# B&R Automation Studio project Lab2_Conveyor (part 2)

### Stations.var - not listed in the package file held
```iecst
VAR
	Conveyor : Conveyor_typ := (Input:=(Par:=(Accel:=100.0,Speed:=100.0,Decel:=100.0)));
	Ejector : Ejector_typ; (*Interface for the Ejector Station*)
	SwivelArm : SwivelArm_typ;
END_VAR
```

### Program Logical/Distributing/Machine/Ejector (IEC)

#### Cyclic.ld - Cyclic code
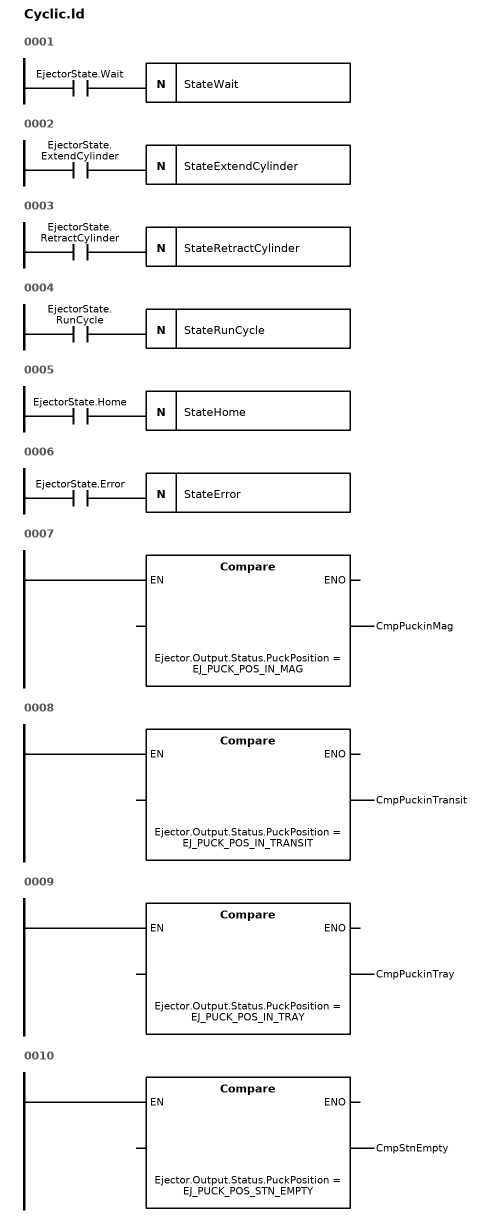
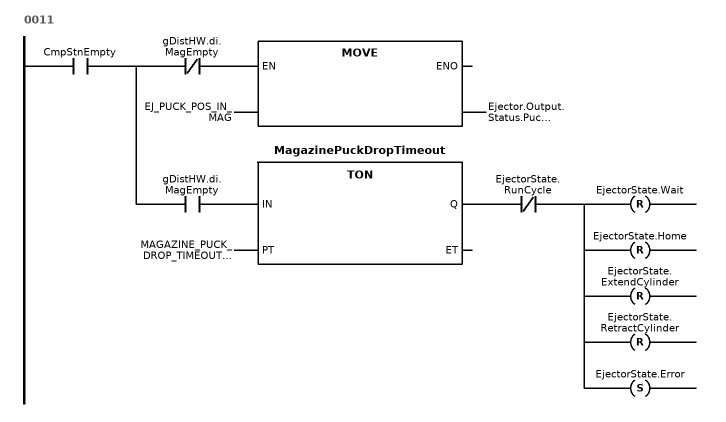
Ladder, written as Structured Text:
```iecst
(*********************************************************************************
 * Copyright: 	B&R Industrial Automation
 * Author:    	Matthew Boyes
 * Created:   	March 8, 2019/12:38 PM
 * Description: 	Task for controlling the operation of the Ejector Station.
 *********************************************************************************)
PROGRAM _CYCLIC
VAR
    _p1 : BOOL;
END_VAR
(* Network 1 *)
IF EjectorState.Wait THEN StateWait; END_IF;

(* Network 2 *)
IF EjectorState.ExtendCylinder THEN StateExtendCylinder; END_IF;

(* Network 3 *)
IF EjectorState.RetractCylinder THEN StateRetractCylinder; END_IF;

(* Network 4 *)
IF EjectorState.RunCycle THEN StateRunCycle; END_IF;

(* Network 5 *)
IF EjectorState.Home THEN StateHome; END_IF;

(* Network 6 *)
IF EjectorState.Error THEN StateError; END_IF;

(* Network 7 *)
CmpPuckinMag := Ejector.Output.Status.PuckPosition = EJ_PUCK_POS_IN_MAG;

(* Network 8 *)
CmpPuckinTransit := Ejector.Output.Status.PuckPosition = EJ_PUCK_POS_IN_TRANSIT;

(* Network 9 *)
CmpPuckinTray := Ejector.Output.Status.PuckPosition = EJ_PUCK_POS_IN_TRAY;

(* Network 10 *)
CmpStnEmpty := Ejector.Output.Status.PuckPosition = EJ_PUCK_POS_STN_EMPTY;

(* Network 11 *)
IF CmpStnEmpty AND NOT gDistHW.di.MagEmpty THEN
    Ejector.Output.Status.PuckPosition := EJ_PUCK_POS_IN_MAG;
END_IF;
MagazinePuckDropTimeout(IN := CmpStnEmpty AND gDistHW.di.MagEmpty, PT := MAGAZINE_PUCK_DROP_TIMEOUT_VALUE);
_p1 := MagazinePuckDropTimeout.Q AND NOT EjectorState.RunCycle;
IF _p1 THEN
    EjectorState.Wait := FALSE;
    EjectorState.Home := FALSE;
    EjectorState.ExtendCylinder := FALSE;
    EjectorState.RetractCylinder := FALSE;
    EjectorState.Error := TRUE;
END_IF;
END_PROGRAM
```

#### Types.typ - Local data types
```iecst
TYPE
	EjectorState_typ : 	STRUCT  (*State machine definition for the Ejector Task*)
		Wait : BOOL := TRUE; (*State in which the Ejector Task is waiting for commands from the MainCtrl Task*)
		RunCycle : BOOL := FALSE; (*State in which the Ejector Task is running a single full operation cycle*)
		ExtendCylinder : BOOL := FALSE; (*State in which the Ejector Task is extending the ejection cylinder in response to a manual command from MainCtrl*)
		RetractCylinder : BOOL := FALSE; (*State in which the Ejector Task is retracting the ejection cylinder in response to a manual command from MainCtrl*)
		Error : BOOL := FALSE; (*Error state for the Ejector Task*)
		Home : BOOL; (*State in which the Ejector Station returns to  it's home position*)
	END_STRUCT;
	EjectorAutoStep_Enum :
		(
		EJECTOR_RETRACT,
		EJECTOR_EXTEND
		);
END_TYPE
```

#### Variables.var - Local variables
```iecst
VAR
	EjectorState : EjectorState_typ;
	CommandProcessing : REFERENCE TO BOOL;
	CylinderExtended : BOOL;
	CylinderRetracted : BOOL;
	AutoStep : EjectorAutoStep_Enum := EJECTOR_EXTEND;
	EjectorExtendTimer : TON;
END_VAR
VAR CONSTANT
	EJECTOR_EXTEND_TIMEOUT : TIME := T#2s;
END_VAR
VAR
	CmpPuckinMag : BOOL;
	CmpPuckinTransit : BOOL;
	CmpPuckinTray : BOOL;
	CmpStnEmpty : BOOL;
	MagazinePuckDropTimeout : TON;
END_VAR
VAR CONSTANT
	MAGAZINE_PUCK_DROP_TIMEOUT_VALUE : TIME := T#1s;
END_VAR
```

#### StateWait.ld
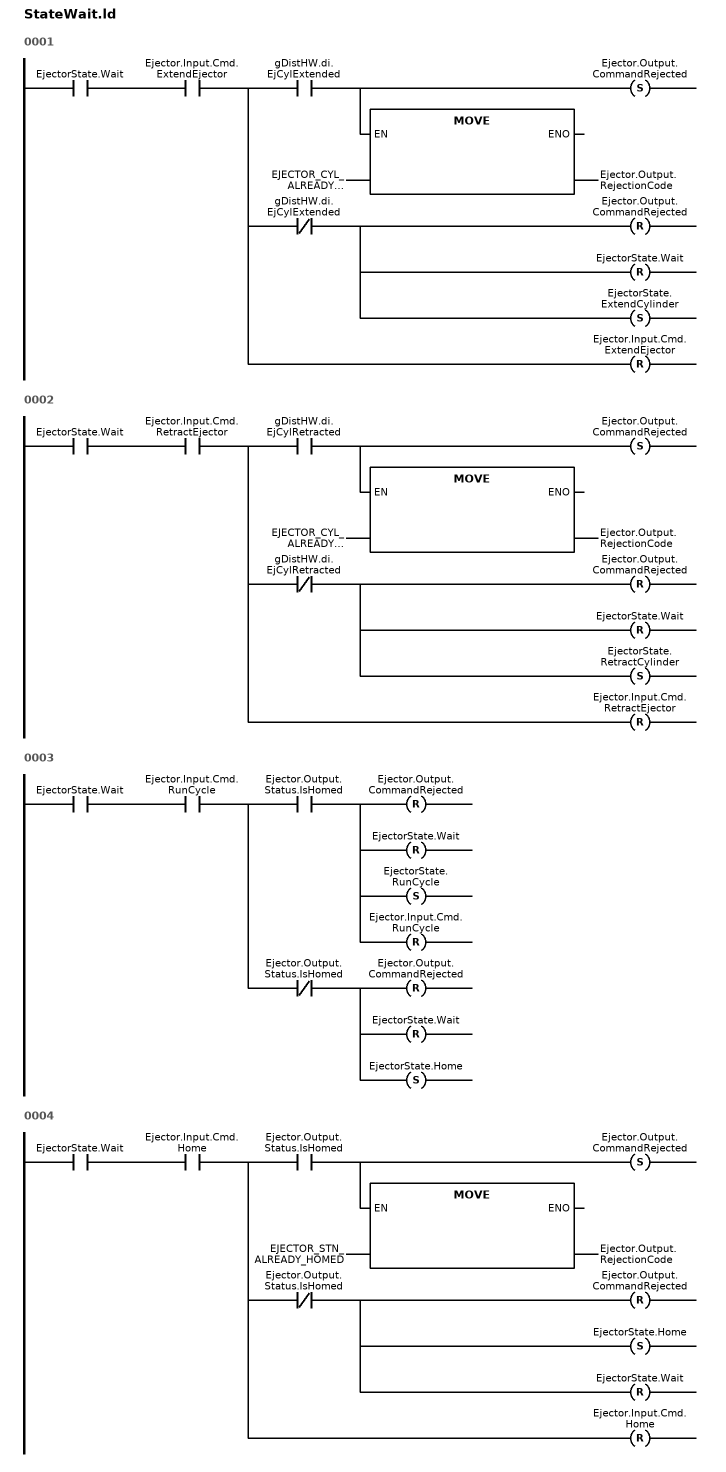
Ladder, written as Structured Text:
```iecst
ACTION StateWait:
VAR
    _p1 : BOOL;
    _p2 : BOOL;
    _p3 : BOOL;
    _p4 : BOOL;
    _p5 : BOOL;
    _p6 : BOOL;
    _p7 : BOOL;
    _p8 : BOOL;
END_VAR
(* Network 1 *)
_p1 := EjectorState.Wait AND Ejector.Input.Cmd.ExtendEjector;
IF _p1 AND gDistHW.di.EjCylExtended THEN
    Ejector.Output.CommandRejected := TRUE;
    Ejector.Output.RejectionCode := EJECTOR_CYL_ALREADY_EXTENDED;
END_IF;
IF _p1 AND NOT gDistHW.di.EjCylExtended THEN
    Ejector.Output.CommandRejected := FALSE;
    EjectorState.Wait := FALSE;
    EjectorState.ExtendCylinder := TRUE;
END_IF;
IF _p1 THEN Ejector.Input.Cmd.ExtendEjector := FALSE; END_IF;

(* Network 2 *)
_p2 := EjectorState.Wait AND Ejector.Input.Cmd.RetractEjector;
IF _p2 AND gDistHW.di.EjCylRetracted THEN
    Ejector.Output.CommandRejected := TRUE;
    Ejector.Output.RejectionCode := EJECTOR_CYL_ALREADY_RETRACTED;
END_IF;
IF _p2 AND NOT gDistHW.di.EjCylRetracted THEN
    Ejector.Output.CommandRejected := FALSE;
    EjectorState.Wait := FALSE;
    EjectorState.RetractCylinder := TRUE;
END_IF;
IF _p2 THEN Ejector.Input.Cmd.RetractEjector := FALSE; END_IF;

(* Network 3 *)
_p3 := EjectorState.Wait AND Ejector.Input.Cmd.RunCycle AND Ejector.Output.Status.IsHomed;
_p4 := EjectorState.Wait AND Ejector.Input.Cmd.RunCycle;
IF _p3 THEN
    Ejector.Output.CommandRejected := FALSE;
    EjectorState.Wait := FALSE;
    EjectorState.RunCycle := TRUE;
    Ejector.Input.Cmd.RunCycle := FALSE;
END_IF;
_p5 := _p4 AND NOT Ejector.Output.Status.IsHomed;
IF _p4 AND NOT Ejector.Output.Status.IsHomed THEN Ejector.Output.CommandRejected := FALSE; END_IF;
IF _p5 THEN
    EjectorState.Wait := FALSE;
    EjectorState.Home := TRUE;
END_IF;

(* Network 4 *)
_p6 := EjectorState.Wait AND Ejector.Input.Cmd.Home AND Ejector.Output.Status.IsHomed;
_p7 := EjectorState.Wait AND Ejector.Input.Cmd.Home;
IF _p6 THEN
    Ejector.Output.CommandRejected := TRUE;
    Ejector.Output.RejectionCode := EJECTOR_STN_ALREADY_HOMED;
END_IF;
_p8 := _p7 AND NOT Ejector.Output.Status.IsHomed;
IF _p7 AND NOT Ejector.Output.Status.IsHomed THEN Ejector.Output.CommandRejected := FALSE; END_IF;
IF _p8 THEN
    EjectorState.Home := TRUE;
    EjectorState.Wait := FALSE;
END_IF;
IF _p7 THEN Ejector.Input.Cmd.Home := FALSE; END_IF;
END_ACTION
```

#### StateExtendCylinder.ld
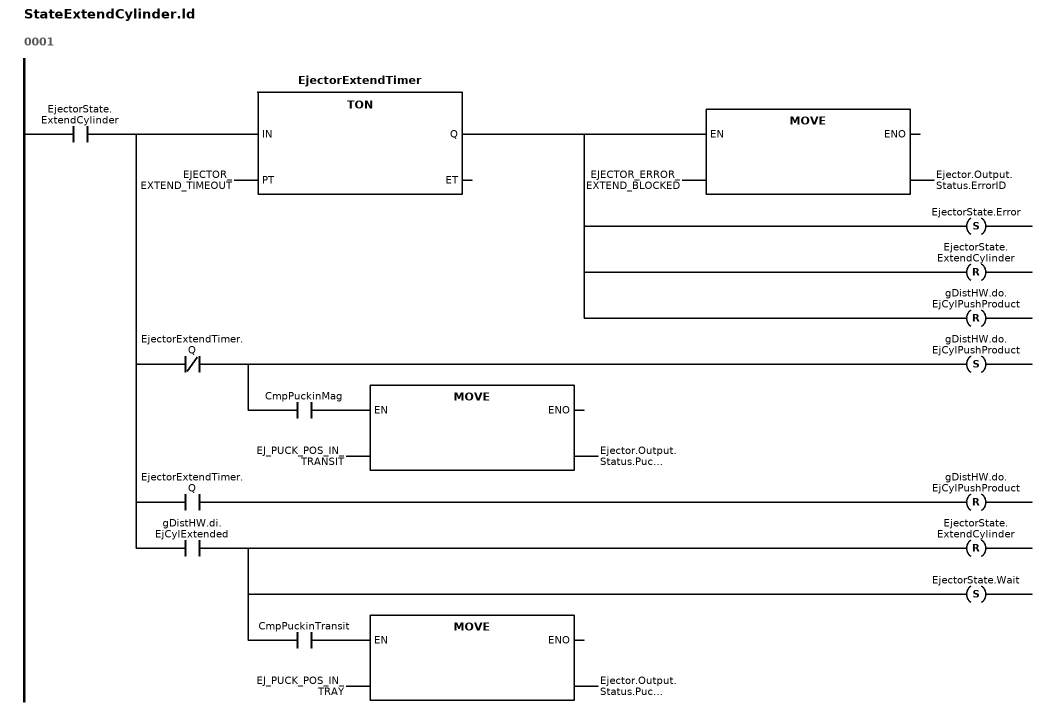
Ladder, written as Structured Text:
```iecst
ACTION StateExtendCylinder:
VAR
    _p1 : BOOL;
END_VAR
(* Network 1 *)
EjectorExtendTimer(IN := EjectorState.ExtendCylinder, PT := EJECTOR_EXTEND_TIMEOUT);
IF EjectorExtendTimer.Q THEN Ejector.Output.Status.ErrorID := EJECTOR_ERROR_EXTEND_BLOCKED; END_IF;
_p1 := EjectorState.ExtendCylinder;
IF EjectorExtendTimer.Q THEN
    EjectorState.Error := TRUE;
    EjectorState.ExtendCylinder := FALSE;
    gDistHW.do.EjCylPushProduct := FALSE;
END_IF;
IF _p1 AND NOT EjectorExtendTimer.Q THEN gDistHW.do.EjCylPushProduct := TRUE; END_IF;
IF _p1 AND NOT EjectorExtendTimer.Q AND CmpPuckinMag THEN
    Ejector.Output.Status.PuckPosition := EJ_PUCK_POS_IN_TRANSIT;
END_IF;
IF _p1 AND EjectorExtendTimer.Q THEN gDistHW.do.EjCylPushProduct := FALSE; END_IF;
IF _p1 AND gDistHW.di.EjCylExtended THEN
    EjectorState.ExtendCylinder := FALSE;
    EjectorState.Wait := TRUE;
END_IF;
IF _p1 AND gDistHW.di.EjCylExtended AND CmpPuckinTransit THEN
    Ejector.Output.Status.PuckPosition := EJ_PUCK_POS_IN_TRAY;
END_IF;
END_ACTION
```

#### StateRetractCylinder.ld
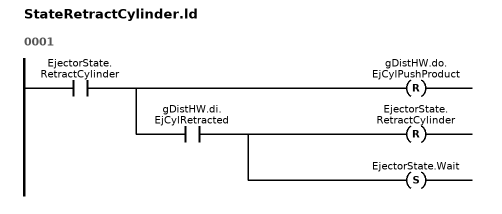
Ladder, written as Structured Text:
```iecst
ACTION StateRetractCylinder:
VAR
    _p1 : BOOL;
END_VAR
(* Network 1 *)
IF EjectorState.RetractCylinder THEN gDistHW.do.EjCylPushProduct := FALSE; END_IF;
_p1 := EjectorState.RetractCylinder AND gDistHW.di.EjCylRetracted;
IF _p1 THEN
    EjectorState.RetractCylinder := FALSE;
    EjectorState.Wait := TRUE;
END_IF;
END_ACTION
```

#### StateRunCycle.ld
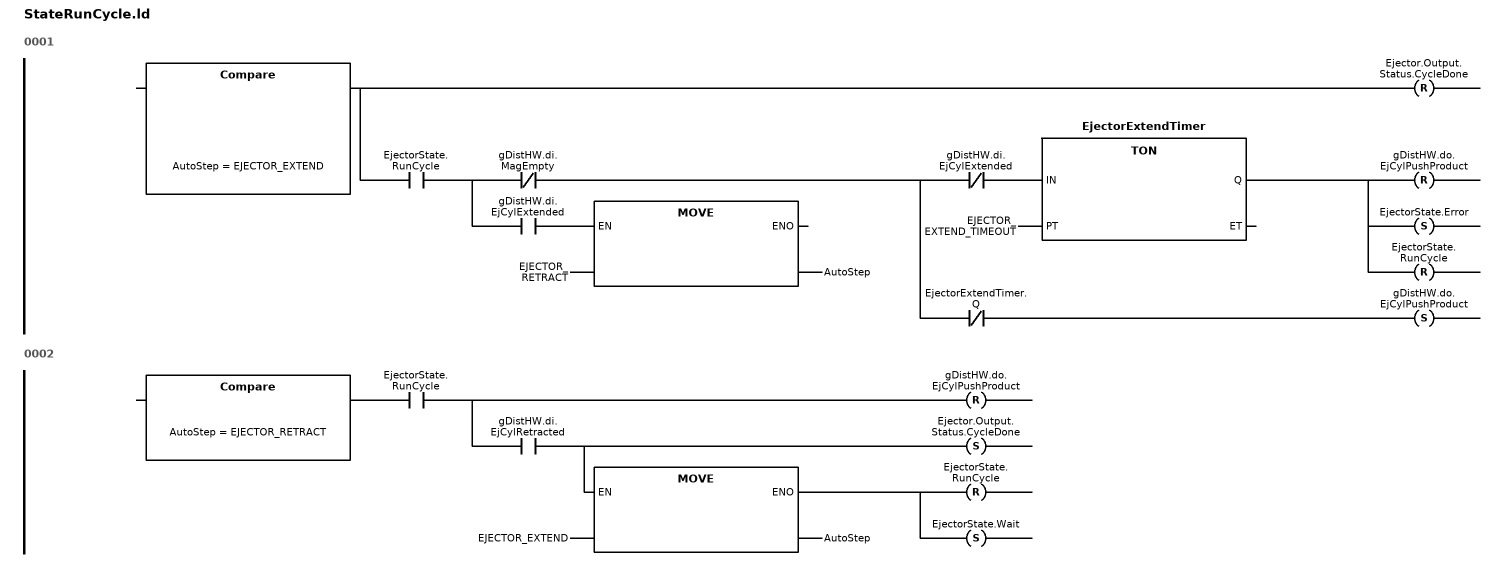
Ladder, written as Structured Text:
```iecst
ACTION StateRunCycle:
VAR
    _p1 : BOOL;
    _p2 : BOOL;
    _p3 : BOOL;
END_VAR
(* Network 1 *)
IF (AutoStep = EJECTOR_EXTEND) THEN Ejector.Output.Status.CycleDone := FALSE; END_IF;
_p1 := (AutoStep = EJECTOR_EXTEND) AND EjectorState.RunCycle;
EjectorExtendTimer(IN := _p1 AND NOT gDistHW.di.MagEmpty AND NOT gDistHW.di.EjCylExtended, PT := EJECTOR_EXTEND_TIMEOUT);
_p2 := _p1 AND NOT gDistHW.di.MagEmpty;
IF EjectorExtendTimer.Q THEN
    gDistHW.do.EjCylPushProduct := FALSE;
    EjectorState.Error := TRUE;
END_IF;
IF _p1 AND gDistHW.di.EjCylExtended THEN AutoStep := EJECTOR_RETRACT; END_IF;
IF EjectorExtendTimer.Q THEN EjectorState.RunCycle := FALSE; END_IF;
IF _p2 AND NOT EjectorExtendTimer.Q THEN gDistHW.do.EjCylPushProduct := TRUE; END_IF;

(* Network 2 *)
_p3 := (AutoStep = EJECTOR_RETRACT) AND EjectorState.RunCycle;
IF _p3 THEN gDistHW.do.EjCylPushProduct := FALSE; END_IF;
IF _p3 AND gDistHW.di.EjCylRetracted THEN
    Ejector.Output.Status.CycleDone := TRUE;
    AutoStep := EJECTOR_EXTEND;
    EjectorState.RunCycle := FALSE;
    EjectorState.Wait := TRUE;
END_IF;
END_ACTION
```

#### StateHome.ld
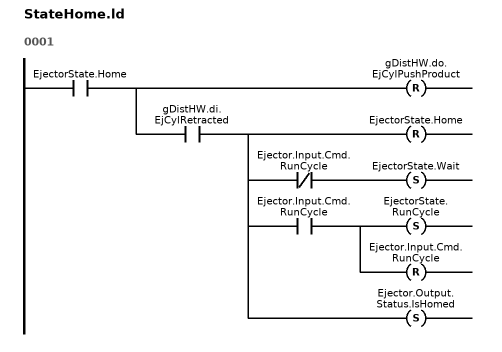
Ladder, written as Structured Text:
```iecst
ACTION StateHome:
VAR
    _p1 : BOOL;
END_VAR
(* Network 1 *)
IF EjectorState.Home THEN gDistHW.do.EjCylPushProduct := FALSE; END_IF;
_p1 := EjectorState.Home AND gDistHW.di.EjCylRetracted;
IF EjectorState.Home AND gDistHW.di.EjCylRetracted THEN EjectorState.Home := FALSE; END_IF;
IF _p1 AND NOT Ejector.Input.Cmd.RunCycle THEN EjectorState.Wait := TRUE; END_IF;
IF _p1 AND Ejector.Input.Cmd.RunCycle THEN
    EjectorState.RunCycle := TRUE;
    Ejector.Input.Cmd.RunCycle := FALSE;
END_IF;
IF _p1 THEN Ejector.Output.Status.IsHomed := TRUE; END_IF;
END_ACTION
```

### Program Logical/Distributing/Machine/IOCtrl

#### Cyclic.ld
Ladder, written as Structured Text:
```iecst
(*********************************************************************************
 * Copyright:
 * Author:
 * Created:   	March 8, 2019/12:38 PM
 * Description:
 *********************************************************************************)
 PROGRAM _CYCLIC
END_PROGRAM
```

### Program Logical/Distributing/Machine/MainCtrl (IEC)

#### Cyclic.ld - Cyclic code
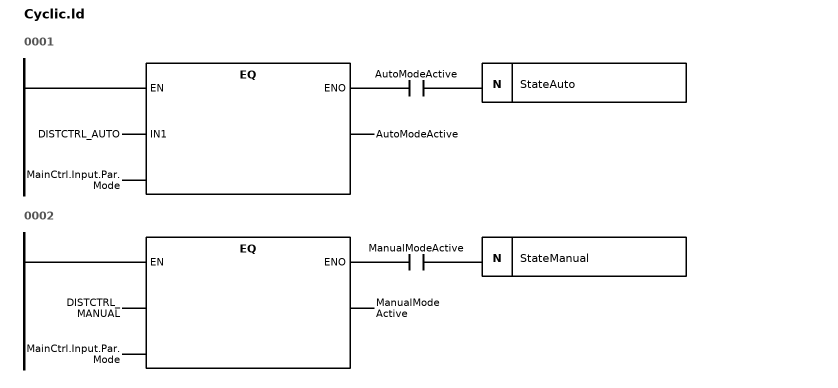
Ladder, written as Structured Text:
```iecst
(*********************************************************************************
 * Copyright:
 * Author:
 * Created:   	March 8, 2019/12:31 PM
 * Description:
 *********************************************************************************)

PROGRAM _CYCLIC
(* Network 1 *)
IF AutoModeActive THEN StateAuto; END_IF;
AutoModeActive := DISTCTRL_AUTO = MainCtrl.Input.Par.Mode;

(* Network 2 *)
IF ManualModeActive THEN StateManual; END_IF;
ManualModeActive := DISTCTRL_MANUAL = MainCtrl.Input.Par.Mode;
END_PROGRAM
```

#### Types.typ - Local data types
```iecst
TYPE
	MainAutoStep_Enum :
		(
		DIST_INIT := 0,
		DIST_CYCLE_EJECTOR := 1,
		DIST_CYCLE_SWIVEL := 2,
		DIST_CYCLE_CONVEYOR := 3,
		DIST_WAIT_FOR_SORT := 4
		);
	PuckPosition_Enum :
		(
		PUCKPOS_IN_MAG := 0,
		PUCKPOS_IN_TRAY := 1,
		PUCKPOS_IN_SWIVEL := 2,
		PUCKPOS_CONV_START := 3,
		PUCKPOS_CONV_MID := 4,
		PUCKPOS_CONV_END := 5
		);
END_TYPE
```

#### Variables.var - Local variables
```iecst
VAR
	AutoModeActive : BOOL;
	ManualModeActive : BOOL;
	AutoModeInitialized : BOOL;
	MainAutoStep : MainAutoStep_Enum := DIST_CYCLE_EJECTOR;
	DispensedPuckTaken : BOOL;
	EjectorStep : BOOL;
	SwivelStep : BOOL;
	PuckPosition : PuckPosition_Enum;
	ConveyorStep : BOOL;
END_VAR
```

#### StateManual.ld
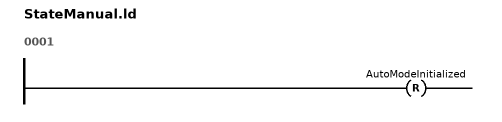
Ladder, written as Structured Text:
```iecst
ACTION StateManual:
(* Network 1 *)
AutoModeInitialized := FALSE;
END_ACTION
```

#### StateAuto.ld
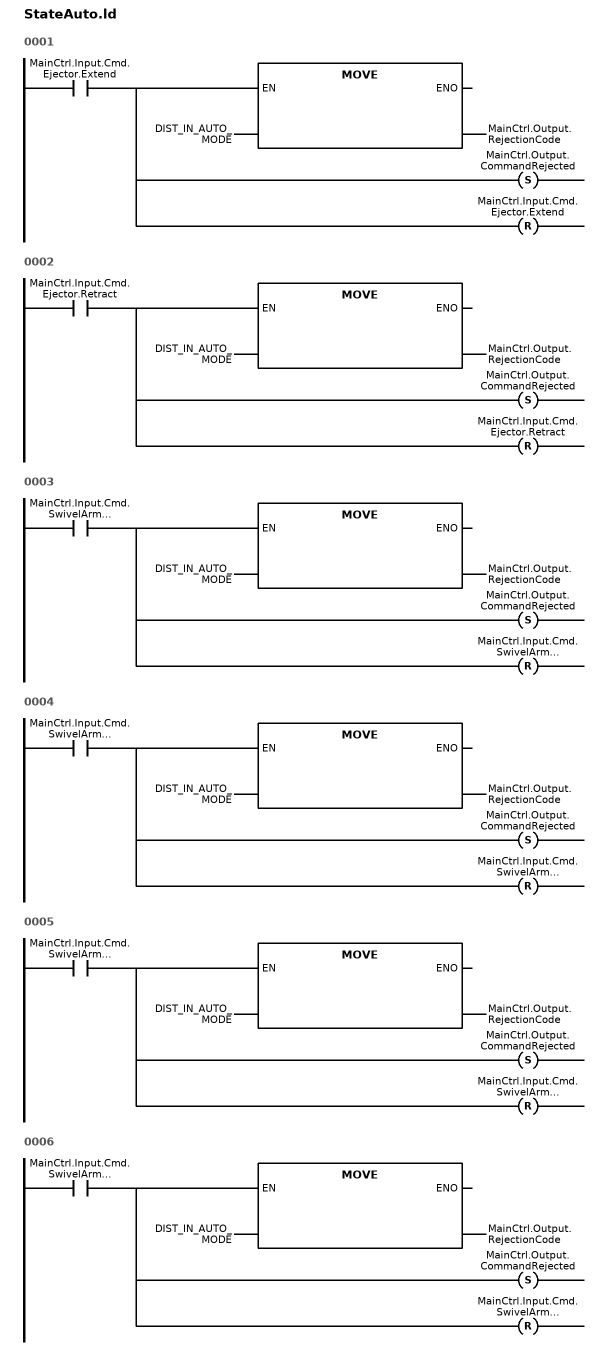
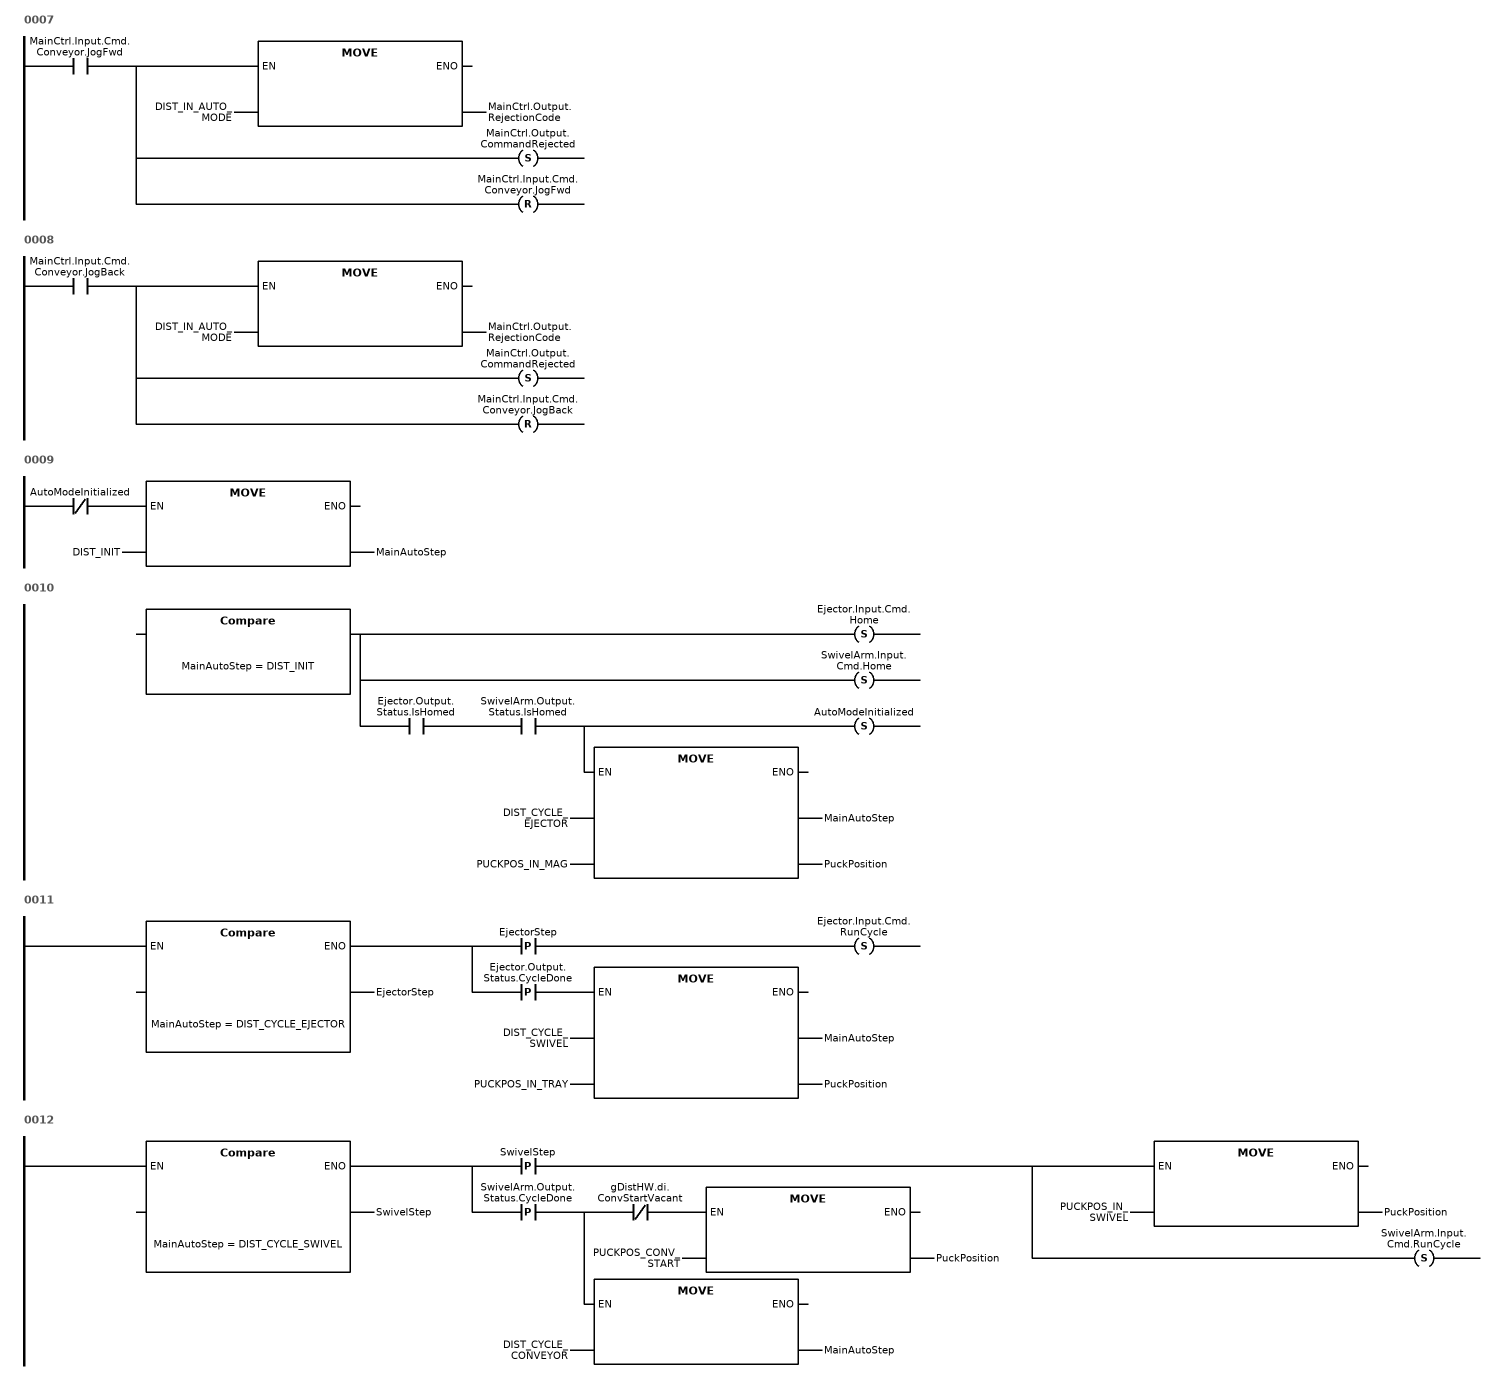
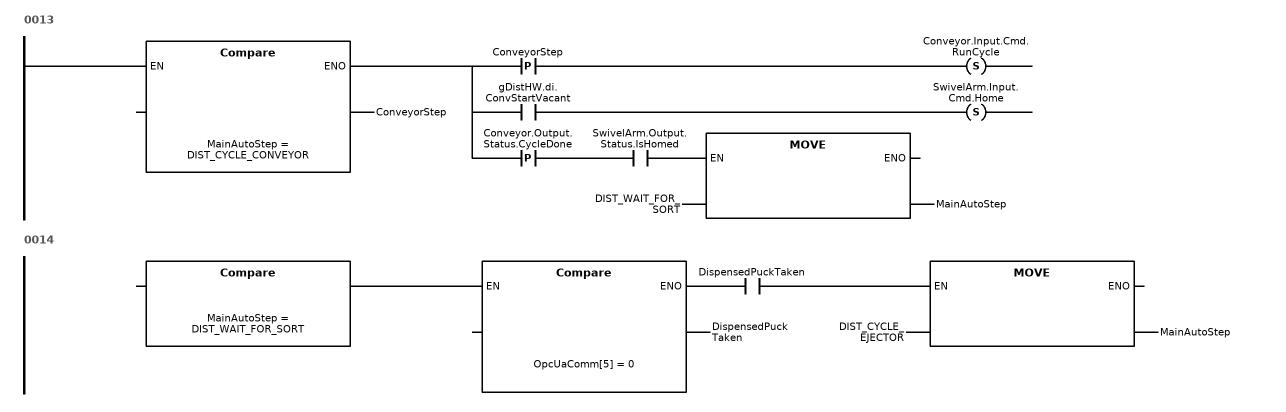
Ladder, written as Structured Text:
```iecst
ACTION StateAuto:
VAR
    _p1 : BOOL;
    _p2 : BOOL;
    _p3 : BOOL;
    _p4 : BOOL;
    _p5 : BOOL;
    _p6 : BOOL;
    _p7 : BOOL;
    _p8 : BOOL;
    _p9 : BOOL;
    _e10 : R_TRIG;
    _e11 : R_TRIG;
    _e12 : R_TRIG;
    _e13 : R_TRIG;
    _e14 : R_TRIG;
    _e15 : R_TRIG;
    _p16 : BOOL;
END_VAR
(* Network 1 *)
_p1 := MainCtrl.Input.Cmd.Ejector.Extend;
IF _p1 THEN
    MainCtrl.Output.RejectionCode := DIST_IN_AUTO_MODE;
    MainCtrl.Output.CommandRejected := TRUE;
    MainCtrl.Input.Cmd.Ejector.Extend := FALSE;
END_IF;

(* Network 2 *)
_p2 := MainCtrl.Input.Cmd.Ejector.Retract;
IF _p2 THEN
    MainCtrl.Output.RejectionCode := DIST_IN_AUTO_MODE;
    MainCtrl.Output.CommandRejected := TRUE;
    MainCtrl.Input.Cmd.Ejector.Retract := FALSE;
END_IF;

(* Network 3 *)
_p3 := MainCtrl.Input.Cmd.SwivelArm.MoveToConveyor;
IF _p3 THEN
    MainCtrl.Output.RejectionCode := DIST_IN_AUTO_MODE;
    MainCtrl.Output.CommandRejected := TRUE;
    MainCtrl.Input.Cmd.SwivelArm.MoveToConveyor := FALSE;
END_IF;

(* Network 4 *)
_p4 := MainCtrl.Input.Cmd.SwivelArm.MoveToMagazine;
IF _p4 THEN
    MainCtrl.Output.RejectionCode := DIST_IN_AUTO_MODE;
    MainCtrl.Output.CommandRejected := TRUE;
    MainCtrl.Input.Cmd.SwivelArm.MoveToMagazine := FALSE;
END_IF;

(* Network 5 *)
_p5 := MainCtrl.Input.Cmd.SwivelArm.VacuumOnImpulse;
IF _p5 THEN
    MainCtrl.Output.RejectionCode := DIST_IN_AUTO_MODE;
    MainCtrl.Output.CommandRejected := TRUE;
    MainCtrl.Input.Cmd.SwivelArm.VacuumOnImpulse := FALSE;
END_IF;

(* Network 6 *)
_p6 := MainCtrl.Input.Cmd.SwivelArm.VacuumOffImpulse;
IF _p6 THEN
    MainCtrl.Output.RejectionCode := DIST_IN_AUTO_MODE;
    MainCtrl.Output.CommandRejected := TRUE;
    MainCtrl.Input.Cmd.SwivelArm.VacuumOffImpulse := FALSE;
END_IF;

(* Network 7 *)
_p7 := MainCtrl.Input.Cmd.Conveyor.JogFwd;
IF _p7 THEN
    MainCtrl.Output.RejectionCode := DIST_IN_AUTO_MODE;
    MainCtrl.Output.CommandRejected := TRUE;
    MainCtrl.Input.Cmd.Conveyor.JogFwd := FALSE;
END_IF;

(* Network 8 *)
_p8 := MainCtrl.Input.Cmd.Conveyor.JogBack;
IF _p8 THEN
    MainCtrl.Output.RejectionCode := DIST_IN_AUTO_MODE;
    MainCtrl.Output.CommandRejected := TRUE;
    MainCtrl.Input.Cmd.Conveyor.JogBack := FALSE;
END_IF;

(* Network 9 *)
IF NOT AutoModeInitialized THEN MainAutoStep := DIST_INIT; END_IF;

(* Network 10 *)
IF (MainAutoStep = DIST_INIT) THEN
    Ejector.Input.Cmd.Home := TRUE;
    SwivelArm.Input.Cmd.Home := TRUE;
END_IF;
_p9 := (MainAutoStep = DIST_INIT) AND Ejector.Output.Status.IsHomed AND SwivelArm.Output.Status.IsHomed;
IF _p9 THEN
    AutoModeInitialized := TRUE;
    MainAutoStep := DIST_CYCLE_EJECTOR;
    PuckPosition := PUCKPOS_IN_MAG;
END_IF;

(* Network 11 *)
_e10(CLK := EjectorStep);
IF _e10.Q THEN Ejector.Input.Cmd.RunCycle := TRUE; END_IF;
EjectorStep := MainAutoStep = DIST_CYCLE_EJECTOR;
_e11(CLK := Ejector.Output.Status.CycleDone);
IF _e11.Q THEN
    MainAutoStep := DIST_CYCLE_SWIVEL;
    PuckPosition := PUCKPOS_IN_TRAY;
END_IF;

(* Network 12 *)
SwivelStep := MainAutoStep = DIST_CYCLE_SWIVEL;
_e12(CLK := SwivelStep);
IF _e12.Q THEN PuckPosition := PUCKPOS_IN_SWIVEL; END_IF;
_e13(CLK := SwivelArm.Output.Status.CycleDone);
IF _e13.Q AND NOT gDistHW.di.ConvStartVacant THEN PuckPosition := PUCKPOS_CONV_START; END_IF;
IF _e12.Q THEN SwivelArm.Input.Cmd.RunCycle := TRUE; END_IF;
IF _e13.Q THEN MainAutoStep := DIST_CYCLE_CONVEYOR; END_IF;

(* Network 13 *)
_e14(CLK := ConveyorStep);
IF _e14.Q THEN Conveyor.Input.Cmd.RunCycle := TRUE; END_IF;
ConveyorStep := MainAutoStep = DIST_CYCLE_CONVEYOR;
IF gDistHW.di.ConvStartVacant THEN SwivelArm.Input.Cmd.Home := TRUE; END_IF;
_e15(CLK := Conveyor.Output.Status.CycleDone);
IF _e15.Q AND SwivelArm.Output.Status.IsHomed THEN MainAutoStep := DIST_WAIT_FOR_SORT; END_IF;

(* Network 14 *)
IF (MainAutoStep = DIST_WAIT_FOR_SORT) THEN DispensedPuckTaken := OpcUaComm[5] = 0; END_IF;
_p16 := (MainAutoStep = DIST_WAIT_FOR_SORT) AND DispensedPuckTaken;
IF _p16 THEN MainAutoStep := DIST_CYCLE_EJECTOR; END_IF;
END_ACTION
```

#### AutoModeHandleManualCmds.ld - not listed in the package file held
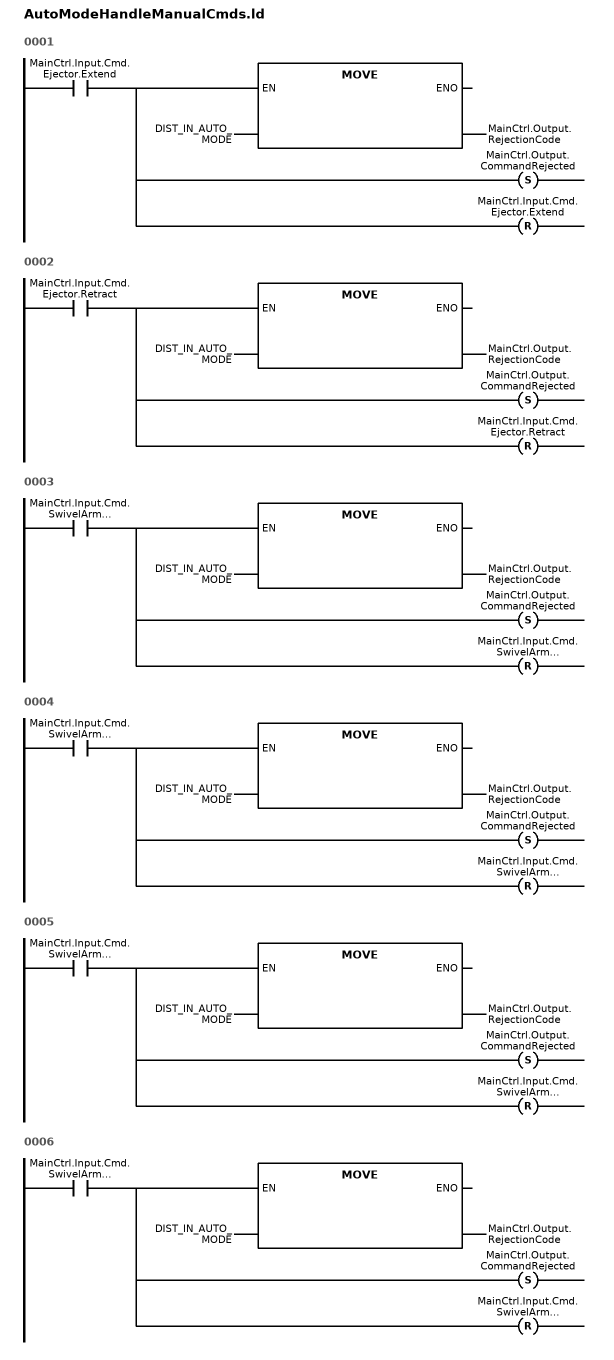
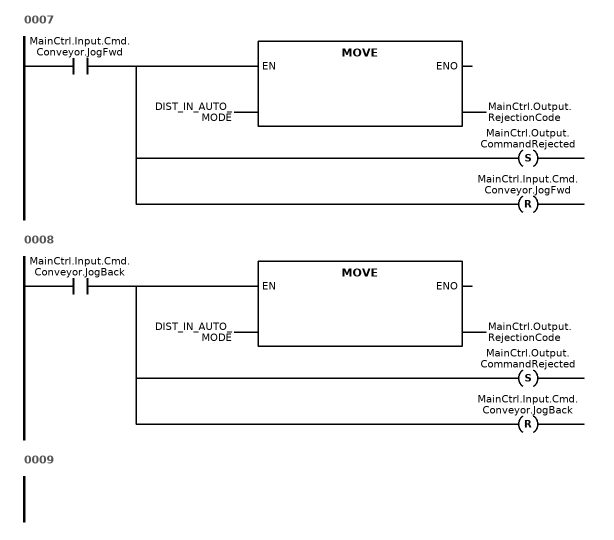
Ladder, written as Structured Text:
```iecst
ACTION AutoModeHandleManualCmds:
VAR
    _p1 : BOOL;
    _p2 : BOOL;
    _p3 : BOOL;
    _p4 : BOOL;
    _p5 : BOOL;
    _p6 : BOOL;
    _p7 : BOOL;
    _p8 : BOOL;
END_VAR
(* Network 1 *)
_p1 := MainCtrl.Input.Cmd.Ejector.Extend;
IF _p1 THEN
    MainCtrl.Output.RejectionCode := DIST_IN_AUTO_MODE;
    MainCtrl.Output.CommandRejected := TRUE;
    MainCtrl.Input.Cmd.Ejector.Extend := FALSE;
END_IF;

(* Network 2 *)
_p2 := MainCtrl.Input.Cmd.Ejector.Retract;
IF _p2 THEN
    MainCtrl.Output.RejectionCode := DIST_IN_AUTO_MODE;
    MainCtrl.Output.CommandRejected := TRUE;
    MainCtrl.Input.Cmd.Ejector.Retract := FALSE;
END_IF;

(* Network 3 *)
_p3 := MainCtrl.Input.Cmd.SwivelArm.MoveToConveyor;
IF _p3 THEN
    MainCtrl.Output.RejectionCode := DIST_IN_AUTO_MODE;
    MainCtrl.Output.CommandRejected := TRUE;
    MainCtrl.Input.Cmd.SwivelArm.MoveToConveyor := FALSE;
END_IF;

(* Network 4 *)
_p4 := MainCtrl.Input.Cmd.SwivelArm.MoveToMagazine;
IF _p4 THEN
    MainCtrl.Output.RejectionCode := DIST_IN_AUTO_MODE;
    MainCtrl.Output.CommandRejected := TRUE;
    MainCtrl.Input.Cmd.SwivelArm.MoveToMagazine := FALSE;
END_IF;

(* Network 5 *)
_p5 := MainCtrl.Input.Cmd.SwivelArm.VacuumOnImpulse;
IF _p5 THEN
    MainCtrl.Output.RejectionCode := DIST_IN_AUTO_MODE;
    MainCtrl.Output.CommandRejected := TRUE;
    MainCtrl.Input.Cmd.SwivelArm.VacuumOnImpulse := FALSE;
END_IF;

(* Network 6 *)
_p6 := MainCtrl.Input.Cmd.SwivelArm.VacuumOffImpulse;
IF _p6 THEN
    MainCtrl.Output.RejectionCode := DIST_IN_AUTO_MODE;
    MainCtrl.Output.CommandRejected := TRUE;
    MainCtrl.Input.Cmd.SwivelArm.VacuumOffImpulse := FALSE;
END_IF;

(* Network 7 *)
_p7 := MainCtrl.Input.Cmd.Conveyor.JogFwd;
IF _p7 THEN
    MainCtrl.Output.RejectionCode := DIST_IN_AUTO_MODE;
    MainCtrl.Output.CommandRejected := TRUE;
    MainCtrl.Input.Cmd.Conveyor.JogFwd := FALSE;
END_IF;

(* Network 8 *)
_p8 := MainCtrl.Input.Cmd.Conveyor.JogBack;
IF _p8 THEN
    MainCtrl.Output.RejectionCode := DIST_IN_AUTO_MODE;
    MainCtrl.Output.CommandRejected := TRUE;
    MainCtrl.Input.Cmd.Conveyor.JogBack := FALSE;
END_IF;

(* Network 9 *)
END_ACTION
```

### Program Logical/Distributing/Machine/SwivelDrive (IEC)

#### Cyclic.ld - Cyclic code
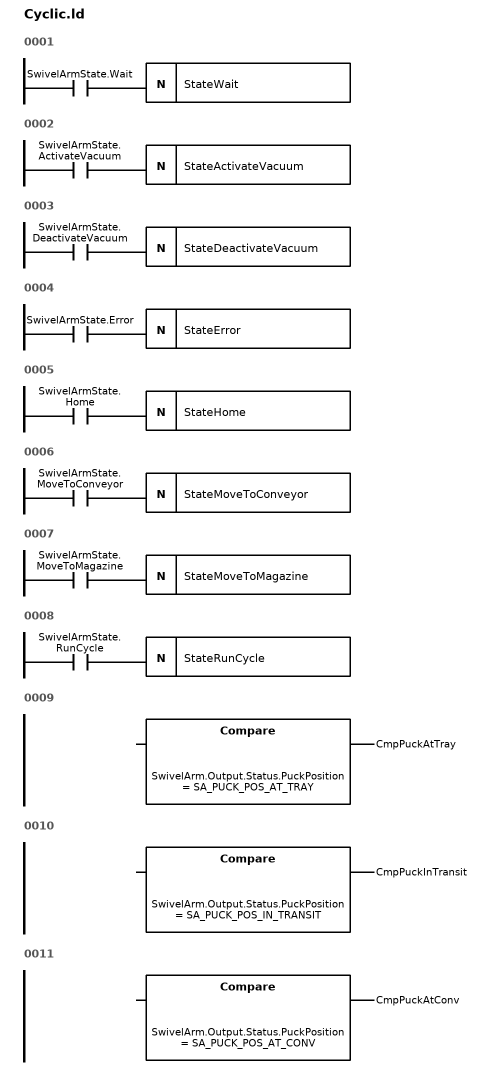
Ladder, written as Structured Text:
```iecst
(*********************************************************************************
 * Copyright: 	B&R Industrial Automation
 * Author:    	Matthew Boyes
 * Created:   	March 8, 2019/12:39 PM
 * Description: 	Controls the swivel arm station.
 *********************************************************************************)
PROGRAM _CYCLIC
(* Network 1 *)
IF SwivelArmState.Wait THEN StateWait; END_IF;

(* Network 2 *)
IF SwivelArmState.ActivateVacuum THEN StateActivateVacuum; END_IF;

(* Network 3 *)
IF SwivelArmState.DeactivateVacuum THEN StateDeactivateVacuum; END_IF;

(* Network 4 *)
IF SwivelArmState.Error THEN StateError; END_IF;

(* Network 5 *)
IF SwivelArmState.Home THEN StateHome; END_IF;

(* Network 6 *)
IF SwivelArmState.MoveToConveyor THEN StateMoveToConveyor; END_IF;

(* Network 7 *)
IF SwivelArmState.MoveToMagazine THEN StateMoveToMagazine; END_IF;

(* Network 8 *)
IF SwivelArmState.RunCycle THEN StateRunCycle; END_IF;

(* Network 9 *)
CmpPuckAtTray := (SwivelArm.Output.Status.PuckPosition = SA_PUCK_POS_AT_TRAY);

(* Network 10 *)
CmpPuckInTransit := (SwivelArm.Output.Status.PuckPosition = SA_PUCK_POS_IN_TRANSIT);

(* Network 11 *)
CmpPuckAtConv := (SwivelArm.Output.Status.PuckPosition = SA_PUCK_POS_AT_CONV);
END_PROGRAM
```

#### Types.typ - Local data types
```iecst
TYPE
	SwivelArmState_typ : 	STRUCT
		Wait : BOOL;
		Home : BOOL;
		DeactivateVacuum : BOOL;
		ActivateVacuum : BOOL;
		MoveToConveyor : BOOL;
		MoveToMagazine : BOOL;
		Error : BOOL;
		RunCycle : BOOL;
	END_STRUCT;
	SwivelAutoStep_Enum :
		(
		MOVE_TO_MAG := 4,
		ACTIVATE_VACUUM := 1,
		MOVE_TO_CONV := 2,
		DEACTIVATE_VACUUM := 3,
		GOTO_PICKUP := 0
		);
END_TYPE
```

#### Variables.var - Local variables
```iecst
VAR
	SwivelArmState : SwivelArmState_typ := (Wait:=TRUE,Home:=FALSE,DeactivateVacuum:=FALSE,ActivateVacuum:=FALSE,MoveToConveyor:=FALSE,MoveToMagazine:=FALSE,Error:=FALSE,RunCycle:=FALSE);
	AutoStep : SwivelAutoStep_Enum := GOTO_PICKUP;
	PickupTimer : TON;
END_VAR
VAR CONSTANT
	PICKUP_TIMER_DELAY : TIME := T#1s;
END_VAR
VAR
	DropoffTimer : TON;
END_VAR
VAR CONSTANT
	DROPOFF_TIMER_DELAY : TIME := T#1s;
END_VAR
VAR
	CmpPuckAtTray : BOOL;
	CmpPuckInTransit : BOOL;
	CmpPuckAtConv : BOOL;
END_VAR
```

#### StateRunCycle.ld
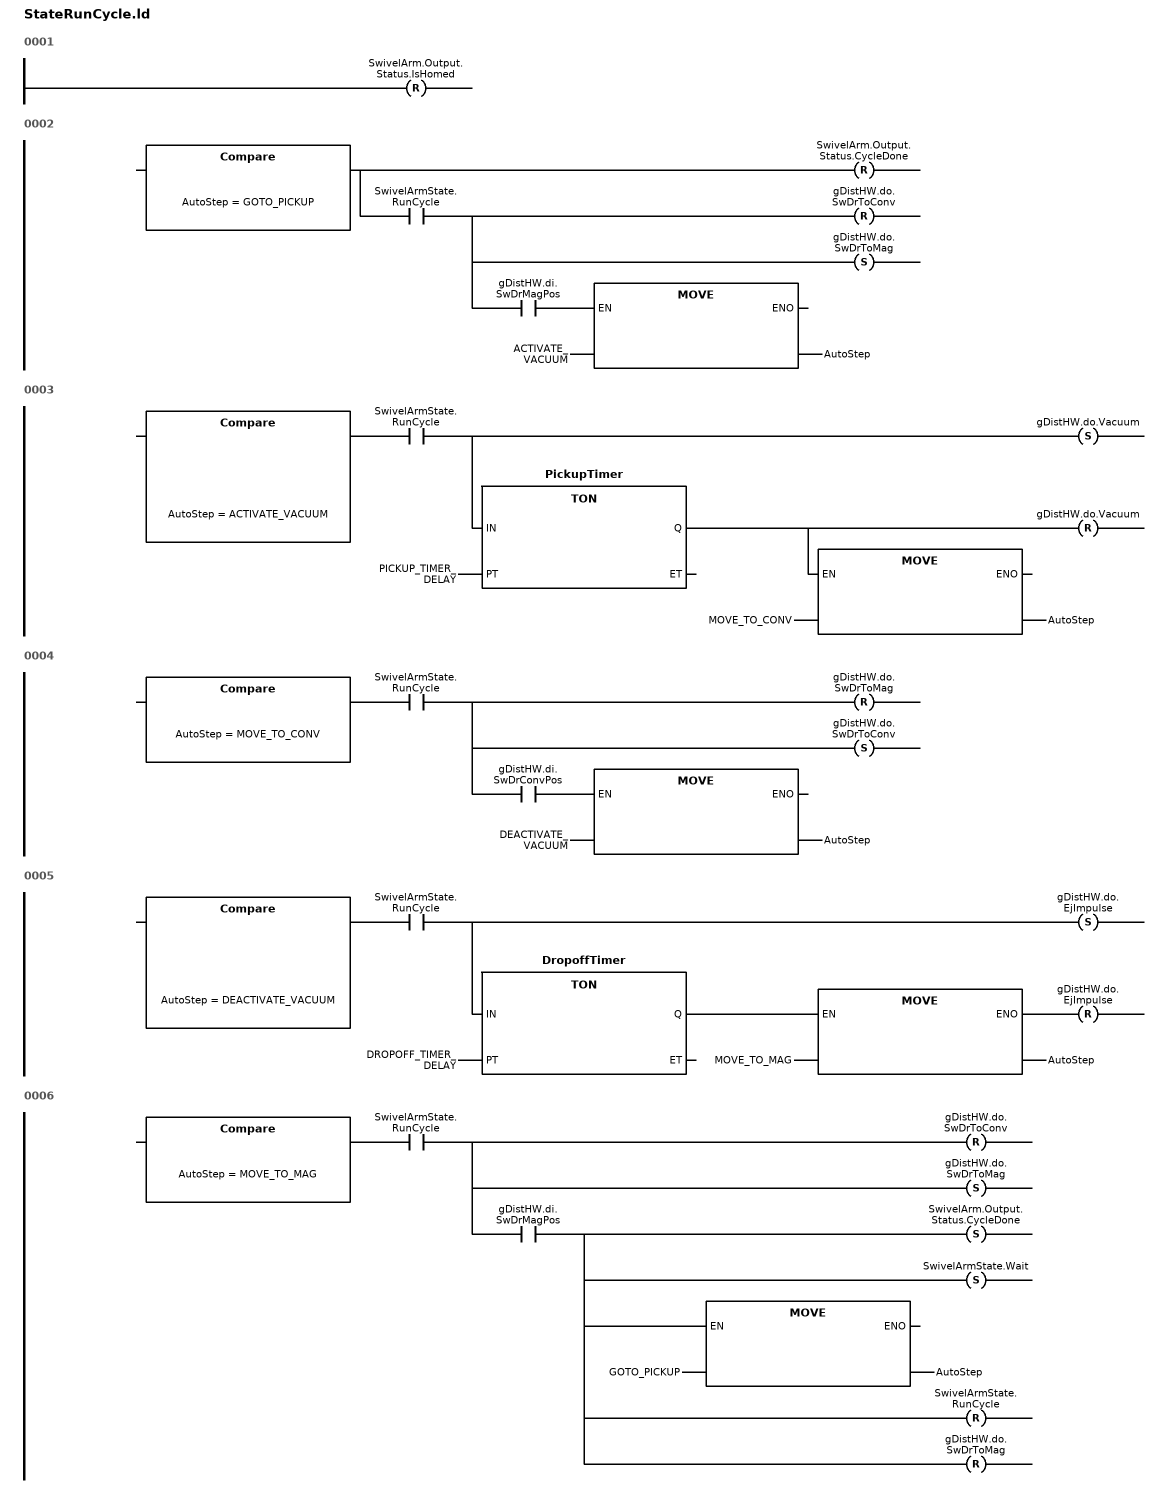
Ladder, written as Structured Text:
```iecst
ACTION StateRunCycle:
VAR
    _p1 : BOOL;
    _p2 : BOOL;
    _p3 : BOOL;
    _p4 : BOOL;
    _p5 : BOOL;
END_VAR
(* Network 1 *)
SwivelArm.Output.Status.IsHomed := FALSE;

(* Network 2 *)
IF (AutoStep = GOTO_PICKUP) THEN SwivelArm.Output.Status.CycleDone := FALSE; END_IF;
_p1 := (AutoStep = GOTO_PICKUP) AND SwivelArmState.RunCycle;
IF _p1 THEN
    gDistHW.do.SwDrToConv := FALSE;
    gDistHW.do.SwDrToMag := TRUE;
END_IF;
IF _p1 AND gDistHW.di.SwDrMagPos THEN AutoStep := ACTIVATE_VACUUM; END_IF;

(* Network 3 *)
_p2 := (AutoStep = ACTIVATE_VACUUM) AND SwivelArmState.RunCycle;
IF _p2 THEN gDistHW.do.Vacuum := TRUE; END_IF;
PickupTimer(IN := _p2, PT := PICKUP_TIMER_DELAY);
IF PickupTimer.Q THEN
    gDistHW.do.Vacuum := FALSE;
    AutoStep := MOVE_TO_CONV;
END_IF;

(* Network 4 *)
_p3 := (AutoStep = MOVE_TO_CONV) AND SwivelArmState.RunCycle;
IF _p3 THEN
    gDistHW.do.SwDrToMag := FALSE;
    gDistHW.do.SwDrToConv := TRUE;
END_IF;
IF _p3 AND gDistHW.di.SwDrConvPos THEN AutoStep := DEACTIVATE_VACUUM; END_IF;

(* Network 5 *)
_p4 := (AutoStep = DEACTIVATE_VACUUM) AND SwivelArmState.RunCycle;
IF _p4 THEN gDistHW.do.EjImpulse := TRUE; END_IF;
DropoffTimer(IN := _p4, PT := DROPOFF_TIMER_DELAY);
IF DropoffTimer.Q THEN
    AutoStep := MOVE_TO_MAG;
    gDistHW.do.EjImpulse := FALSE;
END_IF;

(* Network 6 *)
_p5 := (AutoStep = MOVE_TO_MAG) AND SwivelArmState.RunCycle;
IF _p5 THEN
    gDistHW.do.SwDrToConv := FALSE;
    gDistHW.do.SwDrToMag := TRUE;
END_IF;
IF _p5 AND gDistHW.di.SwDrMagPos THEN
    SwivelArm.Output.Status.CycleDone := TRUE;
    SwivelArmState.Wait := TRUE;
    AutoStep := GOTO_PICKUP;
    SwivelArmState.RunCycle := FALSE;
    gDistHW.do.SwDrToMag := FALSE;
END_IF;
END_ACTION
```

#### StateWait.ld
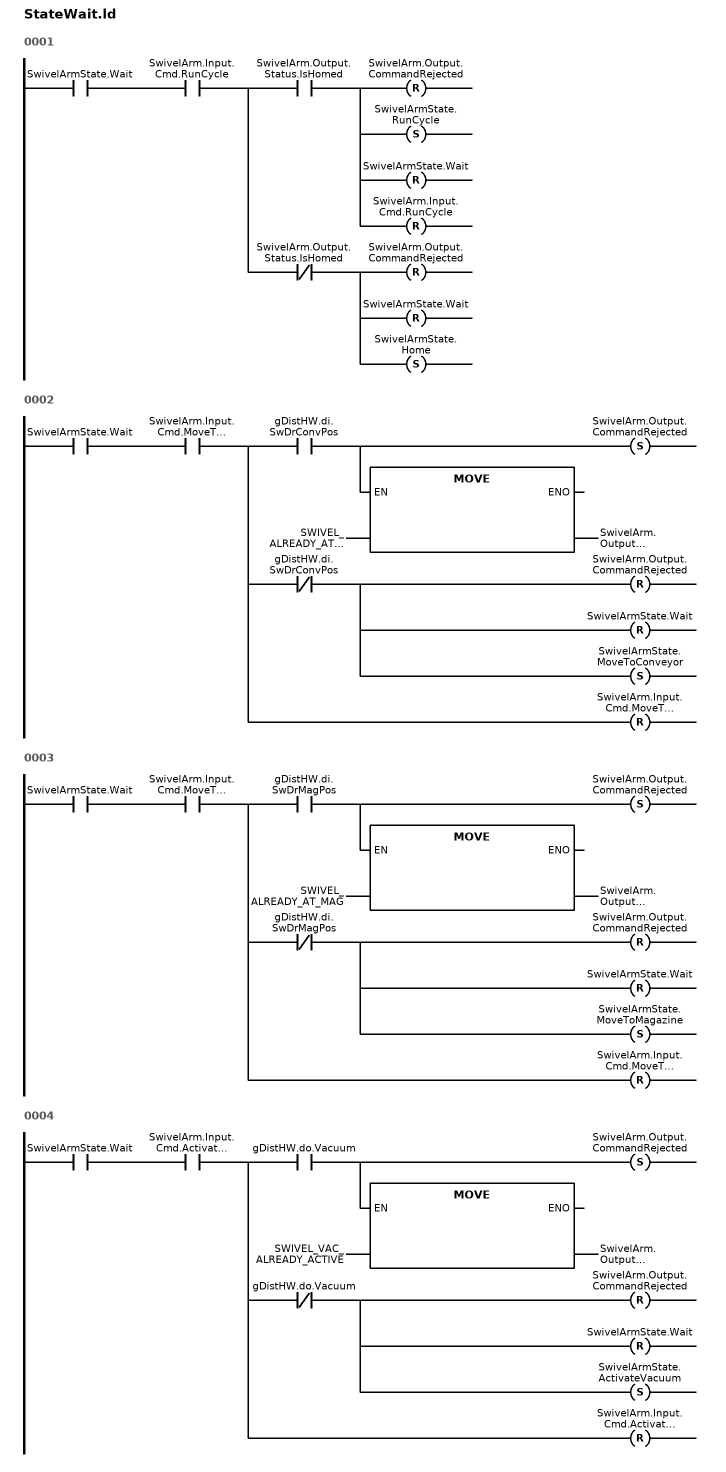
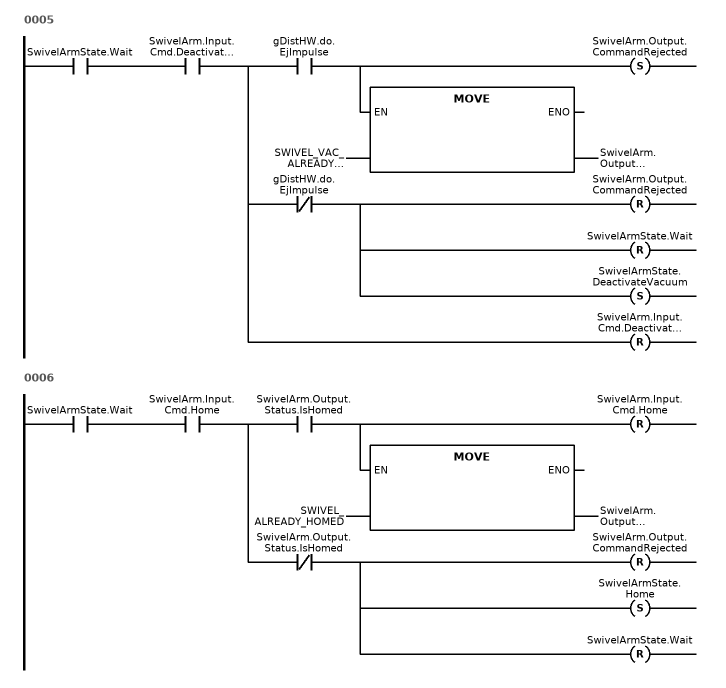
Ladder, written as Structured Text:
```iecst
ACTION StateWait:
VAR
    _p1 : BOOL;
    _p2 : BOOL;
    _p3 : BOOL;
    _p4 : BOOL;
    _p5 : BOOL;
    _p6 : BOOL;
    _p7 : BOOL;
    _p8 : BOOL;
    _p9 : BOOL;
    _p10 : BOOL;
END_VAR
(* Network 1 *)
_p1 := SwivelArmState.Wait AND SwivelArm.Input.Cmd.RunCycle;
_p2 := _p1 AND SwivelArm.Output.Status.IsHomed;
IF _p1 AND SwivelArm.Output.Status.IsHomed THEN SwivelArm.Output.CommandRejected := FALSE; END_IF;
IF _p2 THEN
    SwivelArmState.RunCycle := TRUE;
    SwivelArmState.Wait := FALSE;
    SwivelArm.Input.Cmd.RunCycle := FALSE;
END_IF;
_p3 := _p1 AND NOT SwivelArm.Output.Status.IsHomed;
IF _p1 AND NOT SwivelArm.Output.Status.IsHomed THEN SwivelArm.Output.CommandRejected := FALSE; END_IF;
IF _p3 THEN
    SwivelArmState.Wait := FALSE;
    SwivelArmState.Home := TRUE;
END_IF;

(* Network 2 *)
_p4 := SwivelArmState.Wait AND SwivelArm.Input.Cmd.MoveToConveyor;
IF _p4 AND gDistHW.di.SwDrConvPos THEN
    SwivelArm.Output.CommandRejected := TRUE;
    SwivelArm.Output.RejectionCode := SWIVEL_ALREADY_AT_CONV;
END_IF;
IF _p4 AND NOT gDistHW.di.SwDrConvPos THEN
    SwivelArm.Output.CommandRejected := FALSE;
    SwivelArmState.Wait := FALSE;
    SwivelArmState.MoveToConveyor := TRUE;
END_IF;
IF _p4 THEN SwivelArm.Input.Cmd.MoveToConveyor := FALSE; END_IF;

(* Network 3 *)
_p5 := SwivelArmState.Wait AND SwivelArm.Input.Cmd.MoveToMagazine;
IF _p5 AND gDistHW.di.SwDrMagPos THEN
    SwivelArm.Output.CommandRejected := TRUE;
    SwivelArm.Output.RejectionCode := SWIVEL_ALREADY_AT_MAG;
END_IF;
IF _p5 AND NOT gDistHW.di.SwDrMagPos THEN
    SwivelArm.Output.CommandRejected := FALSE;
    SwivelArmState.Wait := FALSE;
    SwivelArmState.MoveToMagazine := TRUE;
END_IF;
IF _p5 THEN SwivelArm.Input.Cmd.MoveToMagazine := FALSE; END_IF;

(* Network 4 *)
_p6 := SwivelArmState.Wait AND SwivelArm.Input.Cmd.ActivateVacuum;
IF _p6 AND gDistHW.do.Vacuum THEN
    SwivelArm.Output.CommandRejected := TRUE;
    SwivelArm.Output.RejectionCode := SWIVEL_VAC_ALREADY_ACTIVE;
END_IF;
IF _p6 AND NOT gDistHW.do.Vacuum THEN
    SwivelArm.Output.CommandRejected := FALSE;
    SwivelArmState.Wait := FALSE;
    SwivelArmState.ActivateVacuum := TRUE;
END_IF;
IF _p6 THEN SwivelArm.Input.Cmd.ActivateVacuum := FALSE; END_IF;

(* Network 5 *)
_p7 := SwivelArmState.Wait AND SwivelArm.Input.Cmd.DeactivateVacuum;
IF _p7 AND gDistHW.do.EjImpulse THEN
    SwivelArm.Output.CommandRejected := TRUE;
    SwivelArm.Output.RejectionCode := SWIVEL_VAC_ALREADY_INACTIVE;
END_IF;
IF _p7 AND NOT gDistHW.do.EjImpulse THEN
    SwivelArm.Output.CommandRejected := FALSE;
    SwivelArmState.Wait := FALSE;
    SwivelArmState.DeactivateVacuum := TRUE;
END_IF;
IF _p7 THEN SwivelArm.Input.Cmd.DeactivateVacuum := FALSE; END_IF;

(* Network 6 *)
_p8 := SwivelArmState.Wait AND SwivelArm.Input.Cmd.Home AND SwivelArm.Output.Status.IsHomed;
_p9 := SwivelArmState.Wait AND SwivelArm.Input.Cmd.Home;
IF _p8 THEN
    SwivelArm.Input.Cmd.Home := FALSE;
    SwivelArm.Output.RejectionCode := SWIVEL_ALREADY_HOMED;
END_IF;
_p10 := _p9 AND NOT SwivelArm.Output.Status.IsHomed;
IF _p9 AND NOT SwivelArm.Output.Status.IsHomed THEN SwivelArm.Output.CommandRejected := FALSE; END_IF;
IF _p10 THEN
    SwivelArmState.Home := TRUE;
    SwivelArmState.Wait := FALSE;
END_IF;
END_ACTION
```

#### StateActivateVacuum.ld
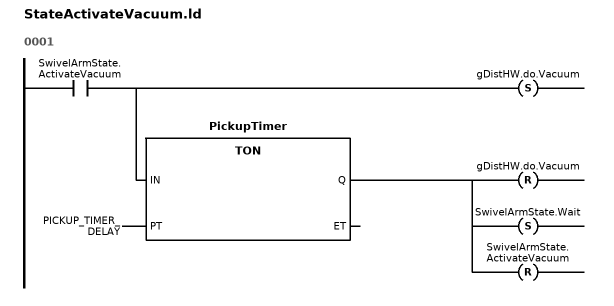
Ladder, written as Structured Text:
```iecst
ACTION StateActivateVacuum:
(* Network 1 *)
IF SwivelArmState.ActivateVacuum THEN gDistHW.do.Vacuum := TRUE; END_IF;
PickupTimer(IN := SwivelArmState.ActivateVacuum, PT := PICKUP_TIMER_DELAY);
IF PickupTimer.Q THEN
    gDistHW.do.Vacuum := FALSE;
    SwivelArmState.Wait := TRUE;
    SwivelArmState.ActivateVacuum := FALSE;
END_IF;
END_ACTION
```

#### StateDeactivateVacuum.ld
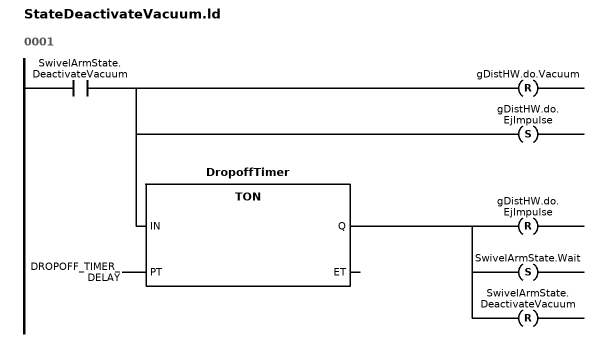
Ladder, written as Structured Text:
```iecst
ACTION StateDeactivateVacuum:
(* Network 1 *)
IF SwivelArmState.DeactivateVacuum THEN
    gDistHW.do.Vacuum := FALSE;
    gDistHW.do.EjImpulse := TRUE;
END_IF;
DropoffTimer(IN := SwivelArmState.DeactivateVacuum, PT := DROPOFF_TIMER_DELAY);
IF DropoffTimer.Q THEN
    gDistHW.do.EjImpulse := FALSE;
    SwivelArmState.Wait := TRUE;
    SwivelArmState.DeactivateVacuum := FALSE;
END_IF;
END_ACTION
```

#### StateHome.ld
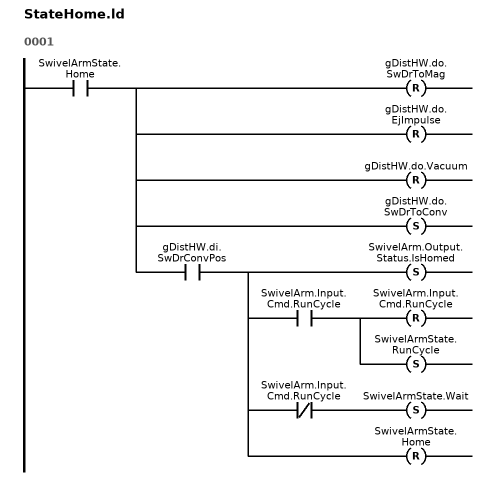
Ladder, written as Structured Text:
```iecst
ACTION StateHome:
VAR
    _p1 : BOOL;
    _p2 : BOOL;
END_VAR
(* Network 1 *)
IF SwivelArmState.Home THEN
    gDistHW.do.SwDrToMag := FALSE;
    gDistHW.do.EjImpulse := FALSE;
    gDistHW.do.Vacuum := FALSE;
    gDistHW.do.SwDrToConv := TRUE;
END_IF;
IF SwivelArmState.Home AND gDistHW.di.SwDrConvPos THEN SwivelArm.Output.Status.IsHomed := TRUE; END_IF;
_p1 := SwivelArmState.Home AND gDistHW.di.SwDrConvPos AND SwivelArm.Input.Cmd.RunCycle;
IF _p1 THEN SwivelArm.Input.Cmd.RunCycle := FALSE; END_IF;
_p2 := SwivelArmState.Home AND gDistHW.di.SwDrConvPos;
IF _p1 THEN SwivelArmState.RunCycle := TRUE; END_IF;
IF _p2 AND NOT SwivelArm.Input.Cmd.RunCycle THEN SwivelArmState.Wait := TRUE; END_IF;
IF _p2 THEN SwivelArmState.Home := FALSE; END_IF;
END_ACTION
```

#### StateMoveToConveyor.ld
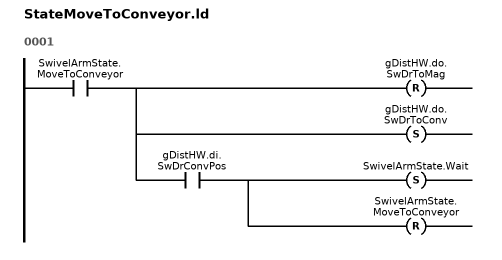
Ladder, written as Structured Text:
```iecst
ACTION StateMoveToConveyor:
VAR
    _p1 : BOOL;
END_VAR
(* Network 1 *)
IF SwivelArmState.MoveToConveyor THEN
    gDistHW.do.SwDrToMag := FALSE;
    gDistHW.do.SwDrToConv := TRUE;
END_IF;
_p1 := SwivelArmState.MoveToConveyor AND gDistHW.di.SwDrConvPos;
IF _p1 THEN
    SwivelArmState.Wait := TRUE;
    SwivelArmState.MoveToConveyor := FALSE;
END_IF;
END_ACTION
```
